FUNCTION_BLOCK BUFFER_196036C8B0617F9B3 (* Generic Buffer Function Block *)
  (* Standard: 61499-2 *)
  (* Version 1.0, 03/07/2019, SESA471741, nxtControl GmbH, initial *)
  PACKAGE UAO.Hackathon;
  (* Compiler Cpp nxtControl builtin 1.0 *)
  {SET_ATTRIBUTE(Runtime.FBType.ImplementingType, Runtime.Standard#DYNGEN_BUFFER)}
  {SET_ATTRIBUTE(Configuration.GenericFBType.InterfaceParams, Runtime.Standard#CNT:=2;DIN${CNT$}:STRING(64),STRING(64))}
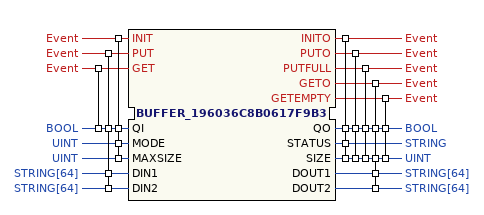
  EVENT_INPUT
    INIT WITH QI, MODE, MAXSIZE; (* Initialize FB clear buffer *)
    PUT WITH QI, DIN1, DIN2; (* Put new DIN into buffer *)
    GET WITH QI; (* Get next DOUT from buffer *)
  END_EVENT
  EVENT_OUTPUT
    INITO WITH QO, STATUS, SIZE; (* INIT done *)
    PUTO WITH QO, SIZE; (* PUT done success *)
    PUTFULL WITH QO, SIZE; (* PUT failed because buffer is full *)
    GETO WITH QO, SIZE, DOUT1, DOUT2; (* GET success *)
    GETEMPTY WITH QO, SIZE; (* GET failed because buffer is empty *)
  END_EVENT
  VAR_INPUT
    QI : BOOL; (* TRUE for normal operation *)
    MODE : UINT; (* 0:FIFO-Queue 1:LIFO-Stack *)
    MAXSIZE : UINT; (* size of preallocated buffer *)
    DIN1 : STRING[64]; (* Input data to buffer *)
    DIN2 : STRING[64]; (* Input data to buffer *)
  END_VAR
  VAR_OUTPUT
    QO : BOOL; (* TRUE for normal operation *)
    STATUS : STRING; (* OK or problem description *)
    SIZE : UINT; (* actual number of buffered elements *)
    DOUT1 : STRING[64]; (* Output data from buffer *)
    DOUT2 : STRING[64]; (* Output data from buffer *)
  END_VAR
  EC_STATES
    START;
  END_STATES
END_FUNCTION_BLOCK
